// Inertface for defining the basic properties of a time instance.
INTERFACE I_TimeInstanceProperties EXTENDS __SYSTEM.IQueryInterface

// The day of the month extracted from the time instance.
// [get] Returns the day component of the date, with a value ranging from 1 to 31.
PROPERTY DayOfMonth : T_DayOfMonth
GET
END_GET
END_PROPERTY

// The day of the week extracted from the time instance.
// [get] Returns the day as an `E_DayOfWeek` enum or value ranging from 1 (Monday) to 7 (Sunday).
PROPERTY DayOfWeek : E_DayOfWeek
GET
END_GET
END_PROPERTY

// The day of the year extracted from the time instance.
// [get] Returns the day of the year, with a value ranging from 1 to 366.
PROPERTY DayOfYear : T_DayOfYear
GET
END_GET
END_PROPERTY

// The time instance value represented as the number of milliseconds since
// Thursday, 1.1.1970 00:00:00.000 (Unix epoch).
// [get] Returns the time instance value in milliseconds.
PROPERTY EpochMilliseconds : ULINT
GET
END_GET
END_PROPERTY

// The hour of the day extracted from the time instance.
// [get] Returns the hour component of the time, with a value ranging from 0 to 23.
PROPERTY Hour : T_Hour
GET
END_GET
END_PROPERTY

// Specifies whether the time instance is in UTC or local time format.
// [get] Returns the time instance type enum as a value.
PROPERTY Kind : E_TimeInstanceKind
GET
END_GET
END_PROPERTY

// The millisecond part of the second extracted from the time instance.
// [get] Returns the millisecond component, with a value ranging from 0 to 999.
PROPERTY Millisecond : T_Millisecond
GET
END_GET
END_PROPERTY

// The minute of the hour extracted from the time instance.
// [get] Returns the minute component, with a value ranging from 0 to 59.
PROPERTY Minute : T_Minute
GET
END_GET
END_PROPERTY

// The month of the year extracted from the time instance.
// [get] Returns the month as an `E_Month` enum or a value ranging from 1 to 12 value.
PROPERTY Month : E_Month
GET
END_GET
END_PROPERTY

// The second of the minute extracted from the time instance.
// [get] Returns the second component, with a value ranging from 0 to 59.
PROPERTY Second : T_Second
GET
END_GET
END_PROPERTY

// The year extracted from the time instance.
// [get] Returns the year as a 4 digit value.
PROPERTY Year : T_Year
GET
END_GET
END_PROPERTY

END_INTERFACE

(* stored: Version 1.1.0.1
   Itf I_TimeInstanceProperties: Id {bdaac79c-e1d3-0683-0d0d-c911bb9719f4}
   Property DayOfMonth: Id {567d3303-c7df-00b7-0535-70b2afb3b710}
   Get Get: Id {ee6a285d-01f9-0bbf-27f3-1b669fb8e5fd}
   Property DayOfWeek: Id {40f80d75-4959-0525-0c05-c8afb8e60be0}
   Get Get: Id {df59ebed-51c9-041b-0939-f8263b3bcdeb}
   Property DayOfYear: Id {64875cc3-db65-0349-29ce-6533ce784f2e}
   Get Get: Id {21dde374-7855-03a3-3411-ed4b73b717f8}
   Property EpochMilliseconds: Id {a071cd63-b602-0095-2c87-22b4d054e579}
   Get Get: Id {c8975830-95b3-0283-0fcc-712e8c8e6f12}
   Property Hour: Id {e59ad18b-4d27-0325-376f-35acd30dc055}
   Get Get: Id {7b200814-1136-0ec2-16ac-c2dc4fff1a79}
   Property Kind: Id {b749c4f1-6711-031a-187b-b04044ad9ac5}
   Get Get: Id {e74488f6-14d9-0284-21e8-d8e03f73405f}
   Property Millisecond: Id {654cc7ae-1ad1-0ffe-1e27-0ce3a0f717ca}
   Get Get: Id {3d09caa9-1db4-0cf3-155c-6dcd71ab8ffe}
   Property Minute: Id {cfabe9f8-1c04-0696-0e30-8ad8f7e2fa4b}
   Get Get: Id {21ab2f68-07aa-04e3-15da-e8a4725cc8f7}
   Property Month: Id {af2ba5d9-ae64-0319-365a-ade27d04bfb8}
   Get Get: Id {efecae49-0d64-0e1b-084d-86c9b881d77c}
   Property Second: Id {94da2a28-8f8a-0d86-218b-0236a8390dbc}
   Get Get: Id {b311cb7b-6995-061f-3e84-e2a4c0eccc0d}
   Property Year: Id {24748c53-8103-0622-2ee6-0a031543f9e3}
   Get Get: Id {a23435a9-bc00-0879-3c7f-00cac728259d} *)
